PROGRAM startup_sequence_prg
VAR
END_VAR

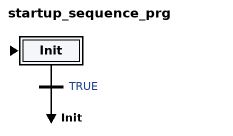
INITIAL_STEP Init:
END_STEP
TRANSITION FROM Init TO Init
    := TRUE;
END_TRANSITION

END_PROGRAM

(* stored: Version 1.1.0.1, ProductVersion 3.1.4024.13
   POU startup_sequence_prg: Id {b12369d1-c148-42fa-8ac0-f7bf6e2ee3c1}, SpecialFunc None *)
